PROGRAM MAIN
VAR
	warmup_sts : FB_State_IOs;
END_VAR

warmup_sts();

END_PROGRAM

(* stored: Version 1.1.0.1, ProductVersion 3.1.4024.12
   POU MAIN: Id {29275dbf-fa6e-414e-9008-085e2326d27d}, SpecialFunc None *)
